// LS Electric XG5000 project: 과년71_3
// PLC NewPLC
// module base 0 slot 0: 입출력 모듈:XBC-DR20S (DC 24V 입력 12점, 릴레이 출력 8점)

PROGRAM NewProgram (task: 스캔 프로그램)

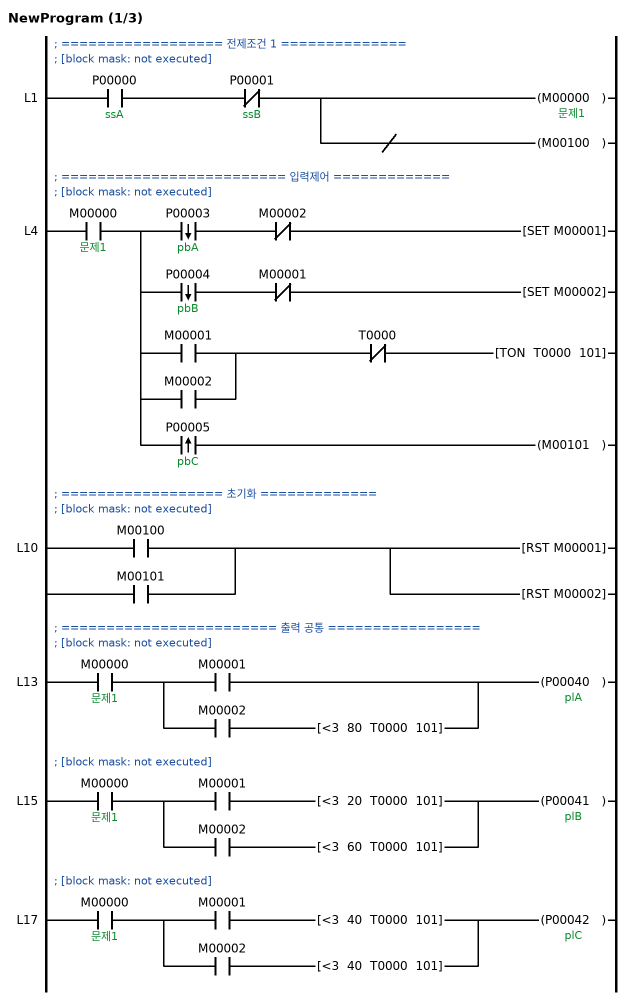
// ================== 전제조건 1 ==============
; L1 (block mask: not executed)
LOAD      P00000	// ssA
AND NOT   P00001	// ssB
OUT       M00000	// 문제1
NOT
OUT       M00100
// ========================= 입력제어 =============
; L4 (block mask: not executed)
LOAD      M00000	// 문제1
MPUSH
ANDN      P00003	// pbA
AND NOT   M00002
SET       M00001
MLOAD
ANDN      P00004	// pbB
AND NOT   M00001
SET       M00002
MLOAD
LOAD      M00001
OR        M00002
AND LOAD
AND NOT   T0000
TON       T0000 101
MPOP
ANDP      P00005	// pbC
OUT       M00101
// ================== 초기화 =============
; L10 (block mask: not executed)
LOAD      M00100
OR        M00101
RST       M00001
RST       M00002
// ======================== 출력 공통 =================
; L13 (block mask: not executed)
LOAD      M00000	// 문제1
LOAD      M00001
LOAD      M00002
AND<3     80 T0000 101
OR LOAD
AND LOAD
OUT       P00040	// plA
; L15 (block mask: not executed)
LOAD      M00000	// 문제1
LOAD      M00001
AND<3     20 T0000 101
LOAD      M00002
AND<3     60 T0000 101
OR LOAD
AND LOAD
OUT       P00041	// plB
; L17 (block mask: not executed)
LOAD      M00000	// 문제1
LOAD      M00001
AND<3     40 T0000 101
LOAD      M00002
AND<3     40 T0000 101
OR LOAD
AND LOAD
OUT       P00042	// plC

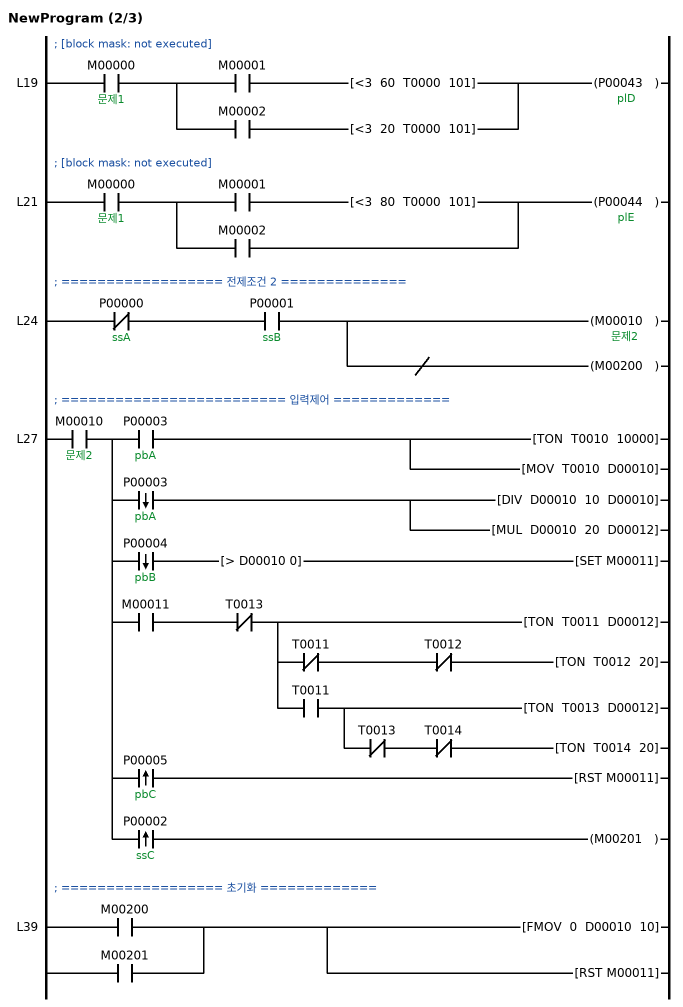
; L19 (block mask: not executed)
LOAD      M00000	// 문제1
LOAD      M00001
AND<3     60 T0000 101
LOAD      M00002
AND<3     20 T0000 101
OR LOAD
AND LOAD
OUT       P00043	// plD
; L21 (block mask: not executed)
LOAD      M00000	// 문제1
LOAD      M00001
AND<3     80 T0000 101
OR        M00002
AND LOAD
OUT       P00044	// plE
// ================== 전제조건 2 ==============
; L24
LOAD NOT  P00000	// ssA
AND       P00001	// ssB
OUT       M00010	// 문제2
NOT
OUT       M00200
// ========================= 입력제어 =============
; L27
LOAD      M00010	// 문제2
MPUSH
AND       P00003	// pbA
TON       T0010 10000
MOV       T0010 D00010
MLOAD
ANDN      P00003	// pbA
DIV       D00010 10 D00010
MUL       D00010 20 D00012
MLOAD
ANDN      P00004	// pbB
AND>      D00010 0
SET       M00011
MLOAD
AND       M00011
AND NOT   T0013
TON       T0011 D00012
MPUSH
AND NOT   T0011
AND NOT   T0012
TON       T0012 20
MPOP
AND       T0011
TON       T0013 D00012
AND NOT   T0013
AND NOT   T0014
TON       T0014 20
MLOAD
ANDP      P00005	// pbC
RST       M00011
MPOP
ANDP      P00002	// ssC
OUT       M00201
// ================== 초기화 =============
; L39
LOAD      M00200
OR        M00201
FMOV      0 D00010 10
RST       M00011

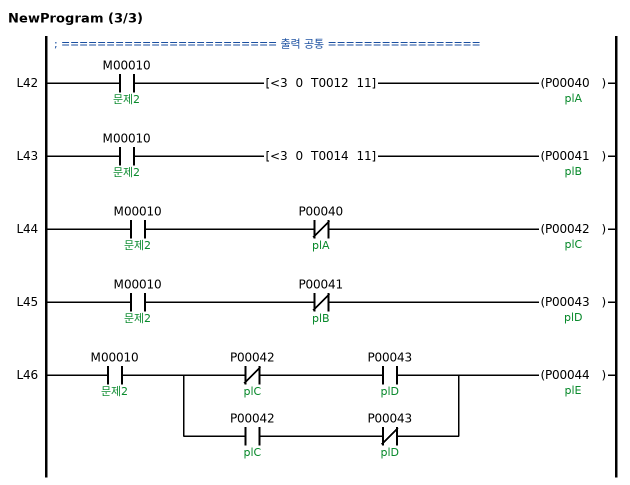
// ======================== 출력 공통 =================
; L42
LOAD      M00010	// 문제2
AND<3     0 T0012 11
OUT       P00040	// plA
; L43
LOAD      M00010	// 문제2
AND<3     0 T0014 11
OUT       P00041	// plB
; L44
LOAD      M00010	// 문제2
AND NOT   P00040	// plA
OUT       P00042	// plC
; L45
LOAD      M00010	// 문제2
AND NOT   P00041	// plB
OUT       P00043	// plD
; L46
LOAD      M00010	// 문제2
LOAD NOT  P00042	// plC
AND       P00043	// plD
LOAD      P00042	// plC
AND NOT   P00043	// plD
OR LOAD
AND LOAD
OUT       P00044	// plE